// TIA Portal V17 export
// export: Created 2024-08-29T18:23:50.7971868Z, ExportSetting WithDefaults, DisplayName Totally Integrated Automation Portal, DisplayVersion V17 Update 7, DisplayName TIA Portal Openness, DisplayVersion V17 Update 7, DisplayName TIA Portal Version Control Interface, DisplayVersion V17, DisplayName SINAMICS Startdrive Advanced, DisplayVersion V17 SP2, DisplayName SINAMICS Startdrive G110M, G120, G120C, G120D, G120P, G115D, DisplayVersion V17 SP2, DisplayName SINAMICS Startdrive G130, G150, S120, S150, SINAMICS MV, S210, DisplayVersion V17 SP2, DisplayName STEP 7 Professional, DisplayVersion V17 Update 7, DisplayName STEP 7 Safety, DisplayVersion V17 Update 6, DisplayName WinCC Advanced / Unified PC, DisplayVersion V17 Update 7
VAR_GLOBAL   // PLC tag table "analogAnalysisMemory"
   leftDistanceOk AT %M1700.4 : Bool;
   rightDistanceOk AT %M1700.5 : Bool;
   leftDistanceOk2 AT %M1700.7 : Bool;
   rightDistanceOk2 AT %M1701.0 : Bool;
   initialAlignmentOK AT %M1700.1 : Bool;
   initialPositionLeftTrackOK AT %M1700.2 : Bool;
   initialPositionRightTrackOK AT %M1700.3 : Bool;
   rightDistanceNormalizedValue AT %MD1660 : Real;
   leftDistanceNormalizedValue AT %MD1664 : Real;
   leftDistanceScaledValue AT %MD1668 : Real;
   rightDistanceScaledValue AT %MD1672 : Real;
   leftEffortOk AT %M1700.0 : Bool;
   rightEffortOk AT %M1700.6 : Bool;
   leftLoadCellSensorValue AT %MW1600 : Int;
   rightLoadCellSensorValue AT %MW1602 : Int;
   leftLoadCellNormalizedValue AT %MD1676 : Real;
   rightLoadCellNormalizedValue AT %MD1680 : Real;
   leftLoadCellScaledValue AT %MD1684 : Real;
   rightLoadCellScaledValue AT %MD1688 : Real;
   leftEffortNok AT %M1701.1 : Bool;
   rightEffortNok AT %M1701.2 : Bool;
   leftTrackRemoveMessage AT %M1701.3 : Bool;
   rightTrackRemoveMessage AT %M1701.4 : Bool;
   leftLoadCellHMIStatus AT %MW1604 : Int;
   rightLoadCellHMIStatus AT %MW1606 : Int;
   leftLoadCellHMIValue AT %MD1692 : Real;
   rightLoadCellHMIValue AT %MD1696 : Real;
END_VAR
